FUNCTION_BLOCK FB_MessageBox
VAR_INPUT
END_VAR
VAR_OUTPUT
END_VAR
VAR
	ID:				ID;
	Message:		STRING(255);
	Arguments:		STRING(255);
END_VAR

END_FUNCTION_BLOCK

(* stored: Version 1.1.0.1
   POU FB_MessageBox: Id {d7235460-dafe-0f48-1a0c-f9a6c027f422}, SpecialFunc None *)
